{attribute 'Tc2GvlVarNames'}
{attribute 'strict'}
//Stato della Missione Della Macchina
TYPE e_Stato_Missione :
(
	NOT_DEFINED									:= -1,
	(*********************************************************************)
	MISSION_STATE_NOP							:= 0,
	(*********************************************************************)
	MISSION_STATE_INIT							:= 10,
	(*********************************************************************)
	MISSION_STATE_VAIaRIPOSO_RUN				:= 20,
	MISSION_STATE_VAIaRIPOSO_END				:= 21,
	(*********************************************************************)
	//MISSION_STATE_PRELIEVO_PALLET_RUN			:= 30,
	//MISSION_STATE_PRELIEVO_PALLET_END			:= 31,
	(*********************************************************************)
	//MISSION_STATE_DEPOSITO_PALLET_RUN			:= 40,
	//MISSION_STATE_DEPOSITO_PALLET_END			:= 41,
	(*********************************************************************)
	MISSION_STATE_PRELIEVO_FALDA_RUN			:= 50,
	MISSION_STATE_PRELIEVO_FALDA_END			:= 51,
	(*********************************************************************)
	MISSION_STATE_DEPOSITO_FALDA_RUN			:= 60,
	MISSION_STATE_DEPOSITO_FALDA_END			:= 61,
	(*********************************************************************)
//	MISSION_STATE_PRELIEVO_PACCO_RUN			:= 70,
	//MISSION_STATE_PRELIEVO_PACCO_END			:= 71,
	(*********************************************************************)
	//MISSION_STATE_DEPOSITO_PACCO_RUN			:= 80,
	//MISSION_STATE_DEPOSITO_PACCO_END			:= 81,
	(*********************************************************************)
	(*********************************************************************)
	
	MISSION_STATE_PRELIEVO_LASTRA_PP_RUN		:= 90,
	MISSION_STATE_PRELIEVO_LASTRA_PP_END		:= 91,
	(*********************************************************************)
	MISSION_STATE_DEPOSITO_LASTRA_PP_RUN		:= 100,
	MISSION_STATE_DEPOSITO_LASTRA_PP_END		:= 101,
	(*********************************************************************)
	MISSION_STATE_PRELIEVO_LASTRA_WA_RUN		:= 110,
	MISSION_STATE_PRELIEVO_LASTRA_WA_END		:= 111,
	(*********************************************************************)
	MISSION_STATE_DEPOSITO_LASTRA_WA_RUN		:= 120,
	MISSION_STATE_DEPOSITO_LASTRA_WA_END		:= 121,
	(*********************************************************************)
	MISSION_STATE_DEPOSITO_LASTRA_SU_PAREGGIATORE_RUN		:= 130,
	MISSION_STATE_DEPOSITO_LASTRA_SU_PAREGGIATORE_END		:= 131,
	(*********************************************************************)
	MISSION_STATE_PAREGGIATURA_RUN		:= 132,
	MISSION_STATE_PAREGGIATURA_END		:= 133,
	(*********************************************************************)
	MISSION_STATE_PRELIEVO_LASTRA_DA_PAREGGIATORE_RUN		:= 134,
	MISSION_STATE_PRELIEVO_LASTRA_DA_PAREGGIATORE_END		:= 135,
	(*********************************************************************)
	MISSION_STATE_PRELIEVO_LASTRA_DEPAL_RUN		:= 136,
	MISSION_STATE_PRELIEVO_LASTRA_DEPAL_END		:= 137,
	(*********************************************************************)
	MISSION_STATE_DEPOSITO_LASTRA_DEPAL_RUN	:= 138,
	MISSION_STATE_DEPOSITO_LASTRA_DEPAL_END	:= 139,
	(*********************************************************************)
	MISSION_STATE_DEPOSITO_FALDA_DEPAL_RUN	:= 140,
	MISSION_STATE_DEPOSITO_FALDA_DEPAL_END	:= 141,
	
	MISSION_STATE_ERROR							:= 999
);
END_TYPE
//  NOT_DEFINED = '-1'

(* stored: Version 1.1.0.1, ProductVersion 3.1.4024.11
   EnumerationTextList e_Stato_Missione: Id {a9cd9038-ffbe-4280-b665-9117a7faa144} *)
